(* Logix 5000 project; controller one_line_prog vendor 1 type 14 code 54 rev 20.19; software revision 20.05 *)

TASK MainTask (continuous, watchdog 500 ms) : MainProgram

MODULES
   Local : vendor 1 type 14 code 54 (ICP 0, rev 20.19)
      OB32_NAMED_AFTER_DISCOVERY : 1756-OB32 (ICP 5, rev 3.2, Output RPI 20 ms)
      OB32_2 : 1756-OB32 (ICP 6, rev 3.2, Output RPI 20 ms)
      IF8 : 1756-IF8 (ICP 7, rev 1.5, Input RPI 100 ms)   // THIS IS IF8 module
END_MODULES

VAR_GLOBAL   (* controller tags *)
   TAG_1_CONT : DINT;
END_VAR

PROGRAM MainProgram   (* main routine MainRoutine *)
VAR
   p_tag_9 : DERIVATIVE := (Gain := 1.0, RTSTime := 1);
   PROG_TAG_5 : BOOL;
   PROG_TAG_5A : DINT;
   PROG_TAG_5B : DINT;
   PROG_TAG_5C : DINT;
   PROG_TAG_5D : DINT;
   PROG_TAG_5E : DINT;
   PROG_TAG_5F : DINT;
   PROG_TAG_5G : DINT;
   PROG_TAG_5H : DINT;
   PROG_TAG_5I : DINT;
   PROG_TAG_5K : DINT;
   PROG_TAG_5L : DINT;
   PROG_TAG_5M : DINT;
   PROG_TAG_5N : DINT;
   PROG_TAG_5O : DINT;
   PROG_TAG_5P : DINT;
   PROG_TAG_5Q : DINT;
   PROG_TAG_5R : DINT;
   PROG_TAG_5S : DINT;
   PROG_TAG_5T : DINT;
   PROG_TAG_5U : DINT;
   PROG_TAG_5V : DINT;
   PROG_TAG_5W : DINT;
   PROG_TAG_5X : DINT;
   PROG_TAG_5Y : DINT;
   PROG_TAG_7 : DERIVATIVE := (Gain := 1.0, RTSTime := 1);
   PROG_TAG_8 : FBD_MATH_ADVANCED;
   PROGRAM_TAG_01 : BOOL;
   PROGRAM_TAG_2 : INT;
   PROGRAM_TAG_4 : INT;
   PROGTAG_3 : BOOL;
   PTAG5A : DINT;
   TAG10 : DINT;
   TAG_6 : BOOL;
END_VAR

ROUTINE MainRoutine   (* ladder *)
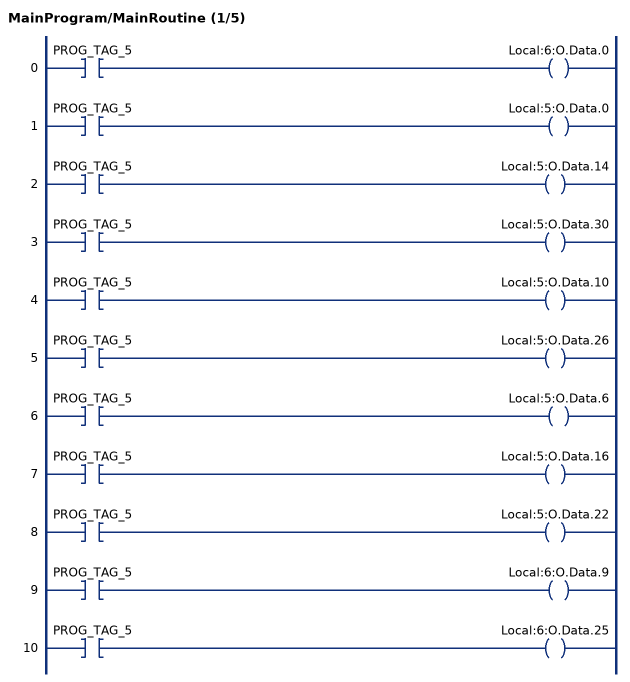
   0: XIC(PROG_TAG_5)OTE(Local:6:O.Data.0);
   1: XIC(PROG_TAG_5)OTE(Local:5:O.Data.0);
   2: XIC(PROG_TAG_5)OTE(Local:5:O.Data.14);
   3: XIC(PROG_TAG_5)OTE(Local:5:O.Data.30);
   4: XIC(PROG_TAG_5)OTE(Local:5:O.Data.10);
   5: XIC(PROG_TAG_5)OTE(Local:5:O.Data.26);
   6: XIC(PROG_TAG_5)OTE(Local:5:O.Data.6);
   7: XIC(PROG_TAG_5)OTE(Local:5:O.Data.16);
   8: XIC(PROG_TAG_5)OTE(Local:5:O.Data.22);
   9: XIC(PROG_TAG_5)OTE(Local:6:O.Data.9);
   10: XIC(PROG_TAG_5)OTE(Local:6:O.Data.25);
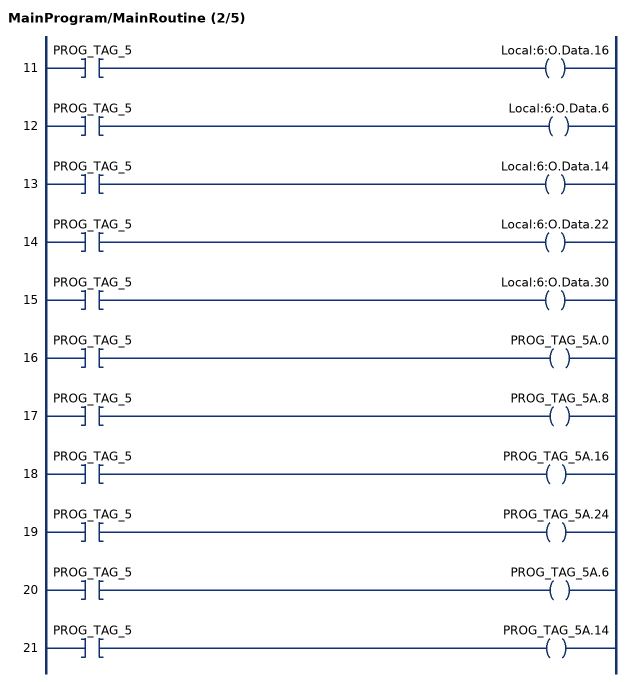
   11: XIC(PROG_TAG_5)OTE(Local:6:O.Data.16);
   12: XIC(PROG_TAG_5)OTE(Local:6:O.Data.6);
   13: XIC(PROG_TAG_5)OTE(Local:6:O.Data.14);
   14: XIC(PROG_TAG_5)OTE(Local:6:O.Data.22);
   15: XIC(PROG_TAG_5)OTE(Local:6:O.Data.30);
   16: XIC(PROG_TAG_5)OTE(PROG_TAG_5A.0);
   17: XIC(PROG_TAG_5)OTE(PROG_TAG_5A.8);
   18: XIC(PROG_TAG_5)OTE(PROG_TAG_5A.16);
   19: XIC(PROG_TAG_5)OTE(PROG_TAG_5A.24);
   20: XIC(PROG_TAG_5)OTE(PROG_TAG_5A.6);
   21: XIC(PROG_TAG_5)OTE(PROG_TAG_5A.14);
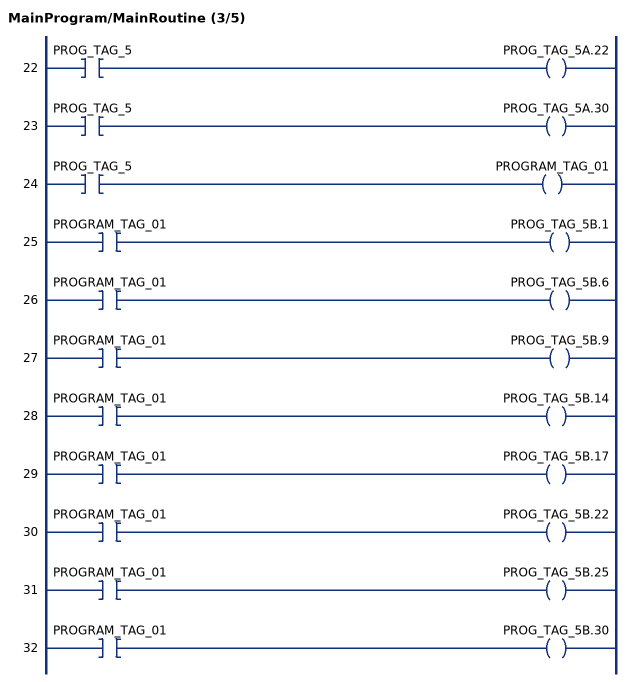
   22: XIC(PROG_TAG_5)OTE(PROG_TAG_5A.22);
   23: XIC(PROG_TAG_5)OTE(PROG_TAG_5A.30);
   24: XIC(PROG_TAG_5)OTE(PROGRAM_TAG_01);
   25: XIC(PROGRAM_TAG_01)OTE(PROG_TAG_5B.1);
   26: XIC(PROGRAM_TAG_01)OTE(PROG_TAG_5B.6);
   27: XIC(PROGRAM_TAG_01)OTE(PROG_TAG_5B.9);
   28: XIC(PROGRAM_TAG_01)OTE(PROG_TAG_5B.14);
   29: XIC(PROGRAM_TAG_01)OTE(PROG_TAG_5B.17);
   30: XIC(PROGRAM_TAG_01)OTE(PROG_TAG_5B.22);
   31: XIC(PROGRAM_TAG_01)OTE(PROG_TAG_5B.25);
   32: XIC(PROGRAM_TAG_01)OTE(PROG_TAG_5B.30);
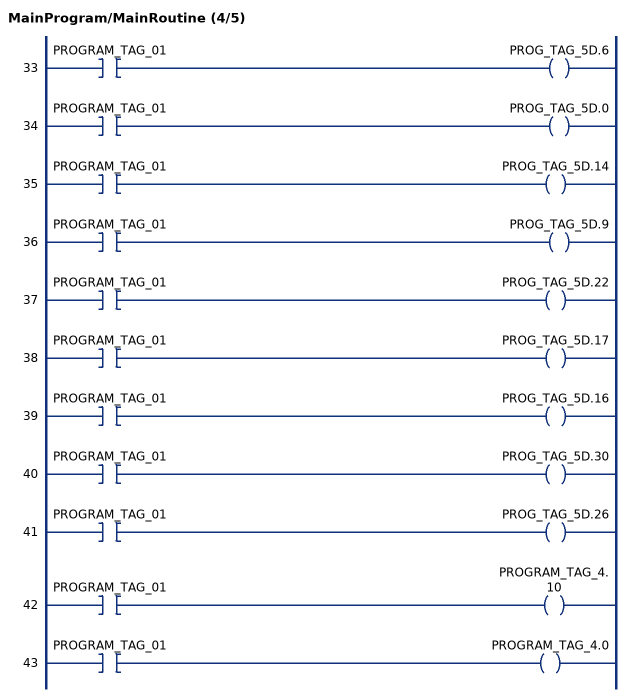
   33: XIC(PROGRAM_TAG_01)OTE(PROG_TAG_5D.6);
   34: XIC(PROGRAM_TAG_01)OTE(PROG_TAG_5D.0);
   35: XIC(PROGRAM_TAG_01)OTE(PROG_TAG_5D.14);
   36: XIC(PROGRAM_TAG_01)OTE(PROG_TAG_5D.9);
   37: XIC(PROGRAM_TAG_01)OTE(PROG_TAG_5D.22);
   38: XIC(PROGRAM_TAG_01)OTE(PROG_TAG_5D.17);
   39: XIC(PROGRAM_TAG_01)OTE(PROG_TAG_5D.16);
   40: XIC(PROGRAM_TAG_01)OTE(PROG_TAG_5D.30);
   41: XIC(PROGRAM_TAG_01)OTE(PROG_TAG_5D.26);
   42: XIC(PROGRAM_TAG_01)OTE(PROGRAM_TAG_4.10);
   43: XIC(PROGRAM_TAG_01)OTE(PROGRAM_TAG_4.0);
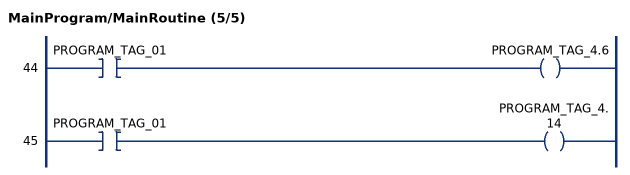
   44: XIC(PROGRAM_TAG_01)OTE(PROGRAM_TAG_4.6);
   45: XIC(PROGRAM_TAG_01)OTE(PROGRAM_TAG_4.14);
END_ROUTINE
END_PROGRAM

PROGRAM PROGRAM2   (* main routine Routine_1_PROG2 *)
VAR
   TAG_1_PROG2 : DINT;
   TAG_2_PROG_2 : DINT;
END_VAR

ROUTINE Routine_1_PROG2   (* ladder *)
END_ROUTINE
END_PROGRAM
